FUNCTION_BLOCK Insertion //2d insertion that combines a slider (alignment) and screw (push)
VAR_INPUT //interface references to existing drives
	slider : I_EncodedDrive;
	screw : I_ContinuousDrive;
END_VAR
VAR_OUTPUT
	contact AT %I* : BOOL;
	
	active : BOOL;
	error : BOOL;
	home : BOOL;
	
	homingComplete : BOOL;
	
	sliderPos : LREAL;
END_VAR
(*
VAR
	slider : LinearDrive_Encoded; //I_PositionalDrive;
	screw : LinearDrive_Continuous; //I_ContinuousDrive;
END_VAR
*)
(*
this FB encapsulates 2 linear drives into a generic insertion machine
both drives should be declared externally in Hardware GVL as a concrete FB
Insertion instance should be declared and called in module scope, with the drives from Hardware GVL passed in by Interface reference
*)

homingComplete := slider.HomeSet AND screw.HomeSet;

active := slider.Active OR screw.Active;
error := slider.Error OR screw.Error;
home := slider.AtHome AND screw.AtHome;

sliderPos := slider.CurrentPosition;

METHOD align : BOOL
VAR_INPUT
	targetPos : REAL;
END_VAR
slider.moveAbsolute(newTarget := targetPos);
END_METHOD

METHOD homingSequence : BOOL
VAR_INPUT
END_VAR
IF NOT slider.homeSet THEN
	slider.homingSequence();
END_IF

IF NOT screw.homeSet THEN
	screw.homingSequence();
END_IF

homingSequence := homingComplete;
END_METHOD

METHOD press : BOOL
VAR_INPUT
END_VAR
IF NOT contact THEN
	screw.moveContinuous(newDirection := MC_Negative_Direction);
END_IF
END_METHOD

METHOD release : BOOL
VAR_INPUT
END_VAR
screw.moveContinuous(newDirection := MC_Positive_Direction);
END_METHOD

METHOD reset : BOOL
VAR_INPUT
END_VAR
slider.reset();
screw.reset();
END_METHOD

METHOD stop : BOOL
VAR_INPUT
END_VAR
screw.stop();
slider.stop();
END_METHOD

METHOD toHome : BOOL
VAR_INPUT
END_VAR
slider.toHome();
screw.toHome();

toHome := slider.AtHome AND screw.AtHome;
END_METHOD

END_FUNCTION_BLOCK

(* stored: Version 1.1.0.1, ProductVersion 3.1.4024.11
   POU Insertion: Id {e64c167d-3486-466f-988e-1abff001b936}, SpecialFunc None
   Method align: Id {3ebc7668-2a9b-443c-a62f-25ae7393caba}
   Method homingSequence: Id {511670a9-8fe8-45d8-baf9-15eef428fd11}
   Method press: Id {c2f6399a-26e3-465f-b5d4-dfbffa94be46}
   Method release: Id {d3f7db45-c06b-4487-9cbc-71279ff85623}
   Method reset: Id {8ee5a51f-b216-4e09-ae47-c041faf0615c}
   Method stop: Id {4e43be39-7934-4202-87dd-4753feeed190}
   Method toHome: Id {fbafc00a-ff70-45ce-b4c3-8537c1253cc3} *)
